INTERFACE I_List

METHOD AddItem : DINT
// Returns the index to which the new object is added into the list,
// or -1  to indicate that the object was not inserted
VAR_INPUT
    ipObject:       I_Object;
END_VAR
END_METHOD

PROPERTY bIsReadOnly : BOOL
GET
END_GET
END_PROPERTY

METHOD Clear
// Remove all items from the list
VAR_INPUT
END_VAR
END_METHOD

METHOD Contains : BOOL
// Determines whether the list contains the querried object
VAR_INPUT
    ipObject:       I_Object;
END_VAR
END_METHOD

METHOD IndexOfItem : DINT
// Returns the zero-based index of the object if it was found in the list,
// otherwise returns -1
VAR_INPUT
    ipObject:       I_Object;
END_VAR
END_METHOD

METHOD Insert : BOOL
// Returns TRUE when object is inserted successfully, and FALSE otherwise
VAR_INPUT
    nIdx:       DINT; // Zero-based index at which object should be inserted
    ipObject:   I_Object; // Object to be inserted
END_VAR
END_METHOD

METHOD ItemAt : I_Object
VAR_INPUT
    nIdx:       DINT;
END_VAR
END_METHOD

PROPERTY nCount : UDINT
GET
END_GET
END_PROPERTY

METHOD Remove
// Remove the first occurerence of a specific object from the list
VAR_INPUT
    ipObject:       I_Object;
END_VAR
END_METHOD

METHOD RemoveAt : BOOL
// Remove an object at the specified index
VAR_INPUT
    nIdx:       DINT;
END_VAR
END_METHOD

END_INTERFACE

(* stored: Version 1.1.0.1, ProductVersion 3.1.4024.12
   Itf I_List: Id {0a9765a5-b03e-0475-3a9d-bcc0b738d24b}
   Method AddItem: Id {84b87bd3-d30a-0279-2a28-36482a97c639}
   Property bIsReadOnly: Id {967d08dc-47ec-0782-07c1-09267a9109a8}
   Get Get: Id {434a0a0c-8d8c-07b6-288b-51788921b9fb}
   Method Clear: Id {fc92d270-56d8-0a15-09d6-6eed49b759a3}
   Method Contains: Id {d530e465-3c8f-0908-2dc5-1716a9b56d2f}
   Method IndexOfItem: Id {cd5c4961-8ca3-07d9-13f3-7aad6fe7ff28}
   Method Insert: Id {11822ce2-2000-0ac2-037d-99062c678a21}
   Method ItemAt: Id {216fb7ca-8a36-0d05-00f7-5a15d03e3914}
   Property nCount: Id {a476dfee-d478-03e7-0628-890d79afb6fb}
   Get Get: Id {9faafaab-84aa-0d3f-032e-bcfc62452ca7}
   Method Remove: Id {9a676453-6f6e-0153-1868-08c54a1da136}
   Method RemoveAt: Id {dc3fb029-e0f1-0053-0870-b3e5e5776683} *)
